Yaskawa INFORM job: TRIG_CAM.JBI

/JOB
//NAME TRIG_CAM
//POS
///NPOS 0,0,0,0,0,0
//INST
///DATE 2022/11/07 11:38
///ATTR SC,RW
///GROUP1 RB1
NOP
TIMER T=1.00
END
